(* Schneider Machine Expert - Basic project Exercise-11 - Multiple Motor Connections with using Set Coil and Normal Coil, file version 2.9.0.0 *)
(* ProjectInformations: Name=New project *)

HARDWARE
  Cpu 0: TM221CE24R
  EthernetConfiguration: NetworkName=M221, IpAllocationMode=FixedAddress, IpAddress=0.0.0.0, SubnetMask=0.0.0.0
  SerialLineConfiguration: Baud=Baud19200, Parity=ParityEven, DataBits=DataBits8, StopBits=StopBits1, PhysicalMedium=PhysicalMediumRs485, SlaveId=1, Addressing=SlaveAddressing
  MastTask: UsePeriodScanMode=false, PeriodScan=100
  FastTask: Period=255
  CpuBehavior: StartingMode=StartAsPreviousState, AutoSaveRamOnEeprom=true, WatchdogPeriod=250

SYMBOLS  (address, symbol, comment, settings)
  %I0.0     SWITCH_1
  %I0.1     SWITCH_2
  %I0.2     SWITCH_3
  %I0.3     SWITCH_4
  %Q0.0     MOTOR_1
  %Q0.1     MOTOR_2
  %Q0.2     MOTOR_3
  %Q0.3     MOTOR_4

POU New POU
  (* SectionNumber=1 *)

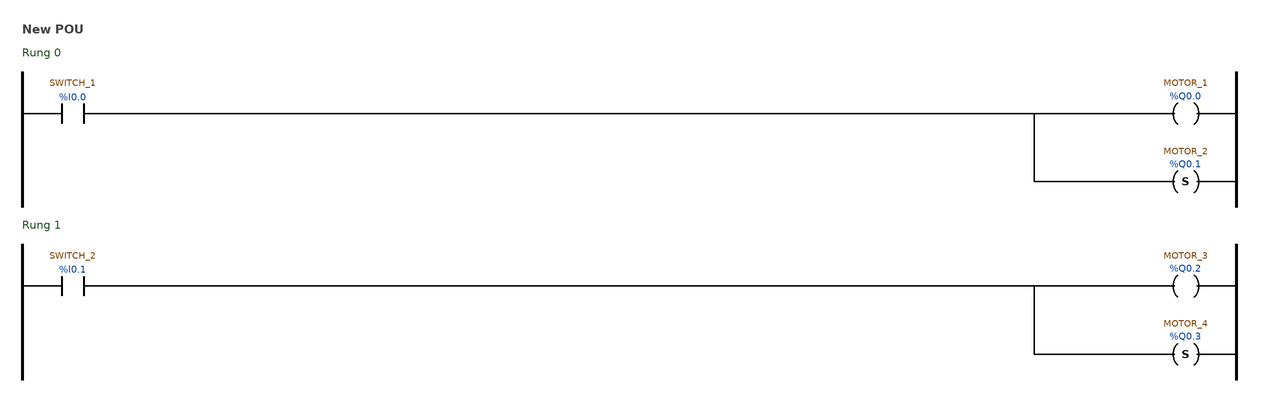

// Rung 0
  LD %I0.0                (* SWITCH_1 *)
  ST %Q0.0                (* MOTOR_1 *)
  S %Q0.1                 (* MOTOR_2 *)
  // as ST:
  //   MOTOR_1 := SWITCH_1;
  //   IF SWITCH_1 THEN MOTOR_2 := TRUE; END_IF;

// Rung 1
  LD %I0.1                (* SWITCH_2 *)
  ST %Q0.2                (* MOTOR_3 *)
  S %Q0.3                 (* MOTOR_4 *)
  // as ST:
  //   MOTOR_3 := SWITCH_2;
  //   IF SWITCH_2 THEN MOTOR_4 := TRUE; END_IF;
